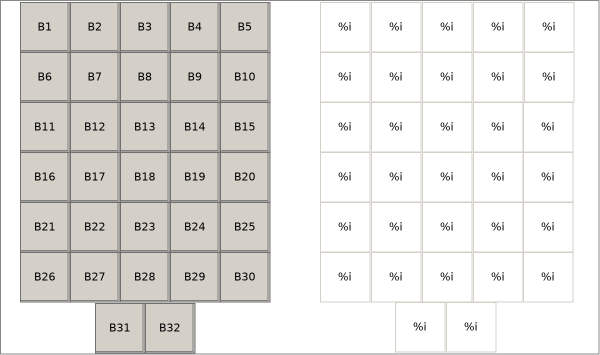
VISUALIZATION Set_Output  // 600x355
    Button (20,2 50x50), "B1", colour toggle: HMI_Global.HMI_OUT_Digital[0]
        toggle HMI_Global.HMI_OUT_Digital[0]
    Textfield (320,2 50x50), "%i", text variable: HMI_Global.HMI_OUT_Analog[0]
        OnMouseDown: write the text variable via VisuDialogs.Numpad, min 0, max 1000
    Button (70,2 50x50), "B2", colour toggle: HMI_Global.HMI_OUT_Digital[1]
        toggle HMI_Global.HMI_OUT_Digital[1]
    Button (120,2 50x50), "B3", colour toggle: HMI_Global.HMI_OUT_Digital[2]
        toggle HMI_Global.HMI_OUT_Digital[2]
    Button (170,2 50x50), "B4", colour toggle: HMI_Global.HMI_OUT_Digital[3]
        toggle HMI_Global.HMI_OUT_Digital[3]
    Button (220,2 50x50), "B5", colour toggle: HMI_Global.HMI_OUT_Digital[4]
        toggle HMI_Global.HMI_OUT_Digital[4]
    Button (20,52 50x50), "B6", colour toggle: HMI_Global.HMI_OUT_Digital[5]
        toggle HMI_Global.HMI_OUT_Digital[5]
    Button (70,52 50x50), "B7", colour toggle: HMI_Global.HMI_OUT_Digital[6]
        toggle HMI_Global.HMI_OUT_Digital[6]
    Button (120,52 50x50), "B8", colour toggle: HMI_Global.HMI_OUT_Digital[7]
        toggle HMI_Global.HMI_OUT_Digital[7]
    Button (170,52 50x50), "B9", colour toggle: HMI_Global.HMI_OUT_Digital[8]
        toggle HMI_Global.HMI_OUT_Digital[8]
    Button (220,52 50x50), "B10", colour toggle: HMI_Global.HMI_OUT_Digital[9]
        toggle HMI_Global.HMI_OUT_Digital[9]
    Button (20,152 50x50), "B16", colour toggle: HMI_Global.HMI_OUT_Digital[15]
        toggle HMI_Global.HMI_OUT_Digital[15]
    Button (20,102 50x50), "B11", colour toggle: HMI_Global.HMI_OUT_Digital[10]
        toggle HMI_Global.HMI_OUT_Digital[10]
    Button (70,102 50x50), "B12", colour toggle: HMI_Global.HMI_OUT_Digital[11]
        toggle HMI_Global.HMI_OUT_Digital[11]
    Button (120,102 50x50), "B13", colour toggle: HMI_Global.HMI_OUT_Digital[12]
        toggle HMI_Global.HMI_OUT_Digital[12]
    Button (170,102 50x50), "B14", colour toggle: HMI_Global.HMI_OUT_Digital[13]
        toggle HMI_Global.HMI_OUT_Digital[13]
    Button (220,102 50x50), "B15", colour toggle: HMI_Global.HMI_OUT_Digital[14]
        toggle HMI_Global.HMI_OUT_Digital[14]
    Button (70,152 50x50), "B17", colour toggle: HMI_Global.HMI_OUT_Digital[16]
        toggle HMI_Global.HMI_OUT_Digital[16]
    Button (120,152 50x50), "B18", colour toggle: HMI_Global.HMI_OUT_Digital[17]
        toggle HMI_Global.HMI_OUT_Digital[17]
    Button (170,152 50x50), "B19", colour toggle: HMI_Global.HMI_OUT_Digital[18]
        toggle HMI_Global.HMI_OUT_Digital[18]
    Button (220,152 50x50), "B20", colour toggle: HMI_Global.HMI_OUT_Digital[19]
        toggle HMI_Global.HMI_OUT_Digital[19]
    Button (20,202 50x50), "B21", colour toggle: HMI_Global.HMI_OUT_Digital[20]
        toggle HMI_Global.HMI_OUT_Digital[20]
    Button (20,252 50x50), "B26", colour toggle: HMI_Global.HMI_OUT_Digital[25]
        toggle HMI_Global.HMI_OUT_Digital[25]
    Button (70,202 50x50), "B22", colour toggle: HMI_Global.HMI_OUT_Digital[21]
        toggle HMI_Global.HMI_OUT_Digital[21]
    Button (120,202 50x50), "B23", colour toggle: HMI_Global.HMI_OUT_Digital[22]
        toggle HMI_Global.HMI_OUT_Digital[22]
    Button (170,202 50x50), "B24", colour toggle: HMI_Global.HMI_OUT_Digital[23]
        toggle HMI_Global.HMI_OUT_Digital[23]
    Button (220,202 50x50), "B25", colour toggle: HMI_Global.HMI_OUT_Digital[24]
        toggle HMI_Global.HMI_OUT_Digital[24]
    Button (70,252 50x50), "B27", colour toggle: HMI_Global.HMI_OUT_Digital[26]
        toggle HMI_Global.HMI_OUT_Digital[26]
    Button (120,252 50x50), "B28", colour toggle: HMI_Global.HMI_OUT_Digital[27]
        toggle HMI_Global.HMI_OUT_Digital[27]
    Button (170,252 50x50), "B29", colour toggle: HMI_Global.HMI_OUT_Digital[28]
        toggle HMI_Global.HMI_OUT_Digital[28]
    Button (220,252 50x50), "B30", colour toggle: HMI_Global.HMI_OUT_Digital[29]
        toggle HMI_Global.HMI_OUT_Digital[29]
    Button (95,303 50x50), "B31", colour toggle: HMI_Global.HMI_OUT_Digital[30]
        toggle HMI_Global.HMI_OUT_Digital[30]
    Button (145,303 50x50), "B32", colour toggle: HMI_Global.HMI_OUT_Digital[31]
        toggle HMI_Global.HMI_OUT_Digital[31]
    Textfield (371,2 50x50), "%i", text variable: HMI_Global.HMI_OUT_Analog[1]
        OnMouseDown: write the text variable via VisuDialogs.Numpad, min 0, max 1000
    Textfield (422,2 50x50), "%i", text variable: HMI_Global.HMI_OUT_Analog[2]
        OnMouseDown: write the text variable via VisuDialogs.Numpad, min 0, max 1000
    Textfield (473,2 50x50), "%i", text variable: HMI_Global.HMI_OUT_Analog[3]
        OnMouseDown: write the text variable via VisuDialogs.Numpad, min 0, max 1000
    Textfield (524,2 50x50), "%i", text variable: HMI_Global.HMI_OUT_Analog[4]
        OnMouseDown: write the text variable via VisuDialogs.Numpad, min 0, max 1000
    Textfield (320,52 50x50), "%i", text variable: HMI_Global.HMI_OUT_Analog[5]
        OnMouseDown: write the text variable via VisuDialogs.Numpad, min 0, max 1000
    Textfield (371,52 50x50), "%i", text variable: HMI_Global.HMI_OUT_Analog[6]
        OnMouseDown: write the text variable via VisuDialogs.Numpad, min 0, max 1000
    Textfield (422,52 50x50), "%i", text variable: HMI_Global.HMI_OUT_Analog[7]
        OnMouseDown: write the text variable via VisuDialogs.Numpad, min 0, max 1000
    Textfield (473,52 50x50), "%i", text variable: HMI_Global.HMI_OUT_Analog[8]
        OnMouseDown: write the text variable via VisuDialogs.Numpad, min 0, max 1000
    Textfield (524,52 50x50), "%i", text variable: HMI_Global.HMI_OUT_Analog[9]
        OnMouseDown: write the text variable via VisuDialogs.Numpad, min 0, max 1000
    Textfield (320,102 50x50), "%i", text variable: HMI_Global.HMI_OUT_Analog[10]
        OnMouseDown: write the text variable via VisuDialogs.Numpad, min 0, max 1000
    Textfield (371,102 50x50), "%i", text variable: HMI_Global.HMI_OUT_Analog[11]
        OnMouseDown: write the text variable via VisuDialogs.Numpad, min 0, max 1000
    Textfield (422,102 50x50), "%i", text variable: HMI_Global.HMI_OUT_Analog[12]
        OnMouseDown: write the text variable via VisuDialogs.Numpad, min 0, max 1000
    Textfield (473,102 50x50), "%i", text variable: HMI_Global.HMI_OUT_Analog[13]
        OnMouseDown: write the text variable via VisuDialogs.Numpad, min 0, max 1000
    Textfield (523,102 50x50), "%i", text variable: HMI_Global.HMI_OUT_Analog[14]
        OnMouseDown: write the text variable via VisuDialogs.Numpad, min 0, max 1000
    Textfield (320,152 50x50), "%i", text variable: HMI_Global.HMI_OUT_Analog[15]
        OnMouseDown: write the text variable via VisuDialogs.Numpad, min 0, max 1000
    Textfield (371,152 50x50), "%i", text variable: HMI_Global.HMI_OUT_Analog[16]
        OnMouseDown: write the text variable via VisuDialogs.Numpad, min 0, max 1000
    Textfield (422,152 50x50), "%i", text variable: HMI_Global.HMI_OUT_Analog[17]
        OnMouseDown: write the text variable via VisuDialogs.Numpad, min 0, max 1000
    Textfield (473,152 50x50), "%i", text variable: HMI_Global.HMI_OUT_Analog[18]
        OnMouseDown: write the text variable via VisuDialogs.Numpad, min 0, max 1000
    Textfield (523,152 50x50), "%i", text variable: HMI_Global.HMI_OUT_Analog[19]
        OnMouseDown: write the text variable via VisuDialogs.Numpad, min 0, max 1000
    Textfield (320,202 50x50), "%i", text variable: HMI_Global.HMI_OUT_Analog[20]
        OnMouseDown: write the text variable via VisuDialogs.Numpad, min 0, max 1000
    Textfield (371,202 50x50), "%i", text variable: HMI_Global.HMI_OUT_Analog[21]
        OnMouseDown: write the text variable via VisuDialogs.Numpad, min 0, max 1000
    Textfield (422,202 50x50), "%i", text variable: HMI_Global.HMI_OUT_Analog[22]
        OnMouseDown: write the text variable via VisuDialogs.Numpad, min 0, max 1000
    Textfield (473,202 50x50), "%i", text variable: HMI_Global.HMI_OUT_Analog[23]
        OnMouseDown: write the text variable via VisuDialogs.Numpad, min 0, max 1000
    Textfield (523,202 50x50), "%i", text variable: HMI_Global.HMI_OUT_Analog[24]
        OnMouseDown: write the text variable via VisuDialogs.Numpad, min 0, max 1000
    Textfield (320,252 50x50), "%i", text variable: HMI_Global.HMI_OUT_Analog[25]
        OnMouseDown: write the text variable via VisuDialogs.Numpad, min 0, max 1000
    Textfield (371,252 50x50), "%i", text variable: HMI_Global.HMI_OUT_Analog[26]
        OnMouseDown: write the text variable via VisuDialogs.Numpad, min 0, max 1000
    Textfield (422,252 50x50), "%i", text variable: HMI_Global.HMI_OUT_Analog[27]
        OnMouseDown: write the text variable via VisuDialogs.Numpad, min 0, max 1000
    Textfield (473,252 50x50), "%i", text variable: HMI_Global.HMI_OUT_Analog[28]
        OnMouseDown: write the text variable via VisuDialogs.Numpad, min 0, max 1000
    Textfield (523,252 50x50), "%i", text variable: HMI_Global.HMI_OUT_Analog[29]
        OnMouseDown: write the text variable via VisuDialogs.Numpad, min 0, max 1000
    Textfield (395,302 50x50), "%i", text variable: HMI_Global.HMI_OUT_Analog[30]
        OnMouseDown: write the text variable via VisuDialogs.Numpad, min 0, max 1000
    Textfield (446,302 50x50), "%i", text variable: HMI_Global.HMI_OUT_Analog[31]
        OnMouseDown: write the text variable via VisuDialogs.Numpad, min 0, max 1000
END_VISUALIZATION

(* stored: Version 1.1.0.1, ProductVersion 3.1.4024.12
   Visu Set_Output: Id {f62a061d-6626-4664-b5f6-9e51efce5e2a} *)
